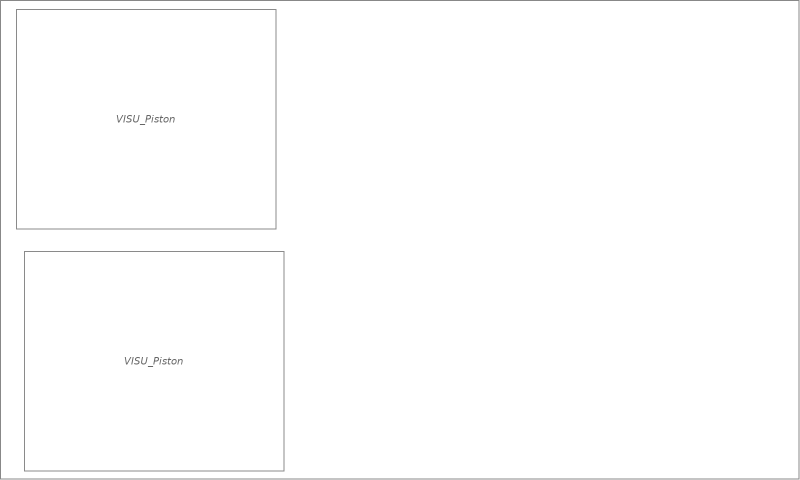
VISUALIZATION VISU_Pistons  // 800x480
    Frame (16,9 260x220)
        shows VISU_Piston(piston := GVL_HMI.stSepSol1)
    Frame (24,251 260x220)
        shows VISU_Piston(piston := GVL_HMI.stPushSol1)
END_VISUALIZATION

(* stored: Version 1.1.0.1, ProductVersion 3.1.4026.18
   Visu VISU_Pistons: Id {cc5c8732-dfa6-4e79-8741-9f75f486b581} *)
